// TwinCAT 3 PLC project GitTrainingRemoveMePlc
// ProgramVersion: 3.1.4023.0
// libraries:
//   Tc2_Standard, * (Beckhoff Automation GmbH)
//   Tc2_System, * (Beckhoff Automation GmbH)
//   Tc2_Utilities, * (Beckhoff Automation GmbH)
//   Tc3_Module, * (Beckhoff Automation GmbH)
// project tree:
//   / PlcTask.TcTTO
//   01_Main/ MAIN.TcPOU
// real-time tasks:
//   TASK PlcTask: cycle T#10ms, priority 20, ADS port 350

CONFIGURATION GitTrainingRemoveMePlc
    RESOURCE PLC ON TwinCAT3
        TASK PlcTask(INTERVAL := T#10ms, PRIORITY := 20);
        PROGRAM MAIN WITH PlcTask : MAIN;
    END_RESOURCE
END_CONFIGURATION

// ---- 01_Main/MAIN.TcPOU
PROGRAM MAIN
VAR
	fbLocalSystemTime			: FB_LocalSystemTime;
END_VAR

IF _TaskInfo[GETCURTASKINDEXEX()].FirstCycle THEN
	fbLocalSystemTime(bEnable := TRUE);
END_IF

fbLocalSystemTime();

END_PROGRAM
